Universal Robots PolyScope program: Program.urp

Program Lab6 (createdIn=3.3.4.310 lastSavedIn=3.3.4.310 directory=/home/ur/ursim-3.3.4.310/programs installation=default robotSerialNumber=2014339999)
Calibrated DH parameters: a=[0.000026, -0.036966, -0.186958, -0.000023, -0.000002, 0]; d=[0.151819, -99.967439, 138.47061, -38.391298, 0.085354, 0.082366]; alpha=[1.57153, -0.002409, -0.002675, 1.571506, -1.571649, 0]; deltaTheta=[0.000018, 1.418493, -1.921964, 0.503527, -0.000019, -0.000014]
Robot Program (runOnlyOnce=false speed=0 acceleration=0 recalculateMotions=false) feature=Base
  URCap
  MoveJ speed 60 deg/s, acceleration 80 deg/s^2 (recalculateMotions=false)
    Waypoint Punto_de_paso_1: TCP in base x=-53.076 y=-383.485 z=316.535 mm, rx=2.8062 ry=0.1005 rz=-0.011 rad; joints [-78.627, -101.549, -32.785, -116.815, 86.444, 726.802] deg; flange x=-53.843 y=-322.378 z=492.833 mm, rx=0.1106 ry=-3.0884 rz=0.5203 rad
  feeder := p[-0.054, -0.5, 0.0435,3.11, 0, 0]
  feeder_up := pose_add(feeder, p[0, 0, 0.05, 0, 0, 0])
  P1 := pose_add(feeder_up, p[0.1, 0.3, 0, 0, 0, 0])
  P2 := pose_add(feeder_up, p[0.2, 0.3, 0, 0, 0, 0])
  P3 := pose_add(feeder_up, p[0.3, 0.3, 0, 0, 0, 0])
  P4 := pose_add(feeder_up, p[0.3, 0.2, 0, 0, 0, 0])
  P5 := pose_add(feeder_up, p[0.3, 0.1, 0, 0, 0, 0])
  P6 := pose_add(feeder_up, p[0.2, 0.1, 0, 0, 0, 0])
  P7 := pose_add(feeder_up, p[0.1, 0.1, 0, 0, 0, 0])
  P8 := pose_add(feeder_up, p[0.1, 0.2, 0, 0, 0, 0])
  P9 := pose_add(feeder_up, p[0.2, 0.2, 0, 0, 0, 0])
  pos := [P1, P2, P3, P4, P5, P6, P7, P8, P9]
  Apieces := [1, 1, 1, 2, 2, 3, 3, 4, 5]
  Loop Counting (count=9) loopVariable(name=Loop_2)
    P := pos[Loop_2]
    pieces := 0
    Pz := pose_add(P, p[0, 0, -0.0473 + (Apieces[Loop_2] - pieces) * 0.02, 0, 0, 0])
    Loop While (checkContinuously=false) expression=pieces≠Apieces[Loop_2]
      MoveJ speed 60 deg/s, acceleration 80 deg/s^2 (recalculateMotions=false)
        Waypoint Punto_de_paso (Variable): variable=feeder
      'Instrucción para agarrar con las pinzas'
      URCap
      MoveJ speed 60 deg/s, acceleration 80 deg/s^2 (recalculateMotions=false)
        Waypoint Punto_de_paso (Variable): variable=feeder_up
      MoveJ speed 60 deg/s, acceleration 80 deg/s^2 (recalculateMotions=false)
        Waypoint Punto_de_paso (Variable): variable=P
      MoveL speed 250 mm/s, acceleration 1200 mm/s^2 (recalculateMotions=false) feature=Base
        Waypoint Punto_de_paso (Variable): variable=Pz
      'Instrucción para soltar'
      URCap
      MoveL speed 250 mm/s, acceleration 1200 mm/s^2 (recalculateMotions=false) feature=Base
        Waypoint Punto_de_paso (Variable): variable=P
      MoveJ speed 60 deg/s, acceleration 80 deg/s^2 (recalculateMotions=false)
        Waypoint Punto_de_paso (Variable): variable=feeder_up
      pieces := pieces + 1
